INTERFACE PUBLIC MoveAbsoluteBuilder EXTENDS __System.IQueryInterface

METHOD PUBLIC Acceleration : MoveAbsoluteBuilder
VAR_INPUT
	value : LREAL;
END_VAR
END_METHOD

METHOD PUBLIC BufferMode : MoveAbsoluteBuilder
VAR_INPUT
	mode : MotionBufferMode;
END_VAR
END_METHOD

METHOD PUBLIC BuildMoveAbsoluteCommand : MotionCommand
VAR_INPUT
	axis : REFERENCE TO Mc2Axis;
END_VAR
END_METHOD

METHOD PUBLIC Deceleration : MoveAbsoluteBuilder
VAR_INPUT
	value : LREAL;
END_VAR
END_METHOD

METHOD PUBLIC Jerk : MoveAbsoluteBuilder
VAR_INPUT
	value : LREAL;
END_VAR
END_METHOD

METHOD PUBLIC Position : MoveAbsoluteBuilder
VAR_INPUT
	value : LREAL;
END_VAR
END_METHOD

METHOD PUBLIC Velocity : MoveAbsoluteBuilder
VAR_INPUT
	value : LREAL;
END_VAR
END_METHOD

END_INTERFACE

(* stored: Version 1.1.0.1
   Itf MoveAbsoluteBuilder: Id {b2204e79-19b1-031b-3f19-69a09b901e25}
   Method Acceleration: Id {39fa12b5-194e-046e-14f0-1d3ab0e70a80}
   Method BufferMode: Id {dfc1ee5e-3b56-09d5-21d4-1b77a02e2a26}
   Method BuildMoveAbsoluteCommand: Id {2e8fdce2-a664-0ca0-1ad6-082fefd9251e}
   Method Deceleration: Id {bbf31b63-5621-0046-3f6a-c1482b4c4e66}
   Method Jerk: Id {6abfc879-829a-02f4-1024-79eef5ad04eb}
   Method Position: Id {199ea2cd-26f7-0b34-043d-6795569072b1}
   Method Velocity: Id {2b5dff68-47b6-0ab5-3c66-a6dee0d95d3a} *)
